FUNCTION_BLOCK INTERNAL FB_Summer EXTENDS FB_SeasonBase
VAR_INPUT
END_VAR
VAR_OUTPUT
END_VAR
VAR
END_VAR

METHOD ChangeToSummerTyres
VAR_INPUT
END_VAR
THIS^._nTyresType := 1;
Tc2_System.ADSLOGSTR(msgCtrlMask := THIS^._nLogLevel,
                     msgFmtStr := 'Changed to summer tyres',
                     strArg := '');
END_METHOD

METHOD FB_init : BOOL
VAR_INPUT
    bInitRetains:           BOOL; // if TRUE, the retain variables are initialized (warm start / cold start)
    bInCopyCode:            BOOL;  // if TRUE, the instance afterwards gets moved into the copy code (online change)
    ipStateMachine:         I_StateMachine;
    ipParentObject:         I_Object;
END_VAR
THIS^._eState := E_Season.Summer;
END_METHOD

METHOD  NextSeason
VAR_INPUT
END_VAR
THIS^.ipStateMachine.SetState(THIS^.ipSeasonCtrl.StateAutumn);
END_METHOD

METHOD OnEntry
SUPER^.OnEntry();
THIS^._bWindBlowing     := FALSE;
THIS^._bRaining         := FALSE;
THIS^._bSunShining      := TRUE;
THIS^._bSnowing         := FALSE;
THIS^._nLeavesState     := 1;
END_METHOD

END_FUNCTION_BLOCK

(* stored: Version 1.1.0.1, ProductVersion 3.1.4024.12
   POU FB_Summer: Id {714eb448-a7ac-09e4-2258-7b0bc36333f9}, SpecialFunc None
   Method ChangeToSummerTyres: Id {9699f616-eee6-080b-1f87-19eac24293bd}
   Method FB_init: Id {4038ee1c-a443-094a-3813-7f061758ce0a}
   Method NextSeason: Id {dd5a8101-9b17-0df1-3365-9a33ecc9e826}
   Method OnEntry: Id {e4310d01-c623-0355-345d-034bd8e442ed} *)
